KUKA KRL program: get_detection.src

&ACCESS RV2
&REL 2
DEFFCT BOOL get_detection(pick_frame: OUT, class: OUT, product: OUT)

   DECL EKI_STATUS ret
   DECL INT status
   DECL FRAME pick_frame
   DECL INT class
   DECL INT product

   status = 3

   ; open network socket
   ret = EKI_Init("get_detection")
   ret = EKI_Open("get_detection")
   WAIT FOR $FLAG[10]

   ; get first frame
   ret = EKI_SetString("get_detection", "request/method", "get_detection")
   ret = EKI_SetString("get_detection", "request/params/representation/type", "string")
   ret = EKI_SetString("get_detection", "request/params/representation/value", "ZYX")
   ret = EKI_SetString("get_detection", "request/params/degrees/type", "bool")
   ret = EKI_SetBool("get_detection", "request/params/degrees/value", TRUE)
   ret = EKI_SetString("get_detection", "request/params/workflow/type", "string")
   ret = EKI_SetString("get_detection", "request/params/workflow/value", "votenet")

   ret = EKI_Send("get_detection", "request")

   WAIT FOR $FLAG[1]
   ret = EKI_GetInt("get_detection","response/status", status)

   ; if there are no get_detections, close socket and return at once
   IF status>0 THEN
      ; close network socket
      ret = EKI_Close("get_detection")
      ret = EKI_Clear("get_detection")
      RETURN FALSE
   ENDIF

   ; parse the received frame
   WAIT FOR $FLAG[2]
   ret = EKI_GetFrame("get_detection","response/params/param/pose", pick_frame)

   ; KUKA poses are in mm
   pick_frame.X = pick_frame.X * 1000
   pick_frame.Y = pick_frame.Y * 1000
   pick_frame.Z = pick_frame.Z * 1000

   ; parse the received class
   WAIT FOR $FLAG[3]
   ret = EKI_GetInt("get_detection","response/params/param/class", class)

   ; parse the received product
   WAIT FOR $FLAG[4]
   ret = EKI_GetInt("get_detection","response/params/param/product", product)

   ; close network socket
   ret = EKI_Close("get_detection")
   ret = EKI_Clear("get_detection")

   RETURN TRUE

ENDFCT
